{attribute addProperty BoxType "AX8810-0000-0017"}
{attribute addProperty Id "StatuswordAT %I*Statusword_3E16C5AB162"}
{attribute addProperty CRC "2958492027"}
{attribute addProperty SizeInBites "16"}
{attribute addProperty SizeInBytes "2"}
TYPE PSM_Statusword_B057017B :
STRUCT
	{attribute addProperty Name "Statusword"}
	Statusword AT %I* : Statusword_3E16C5AB;
END_STRUCT
END_TYPE

(* stored: Version 1.2.0.0, ProductVersion 3.1.4024.9
   DUT PSM_Statusword_B057017B: Id {869d783e-dff6-4bcd-bdc2-022055f2dbd5} *)
